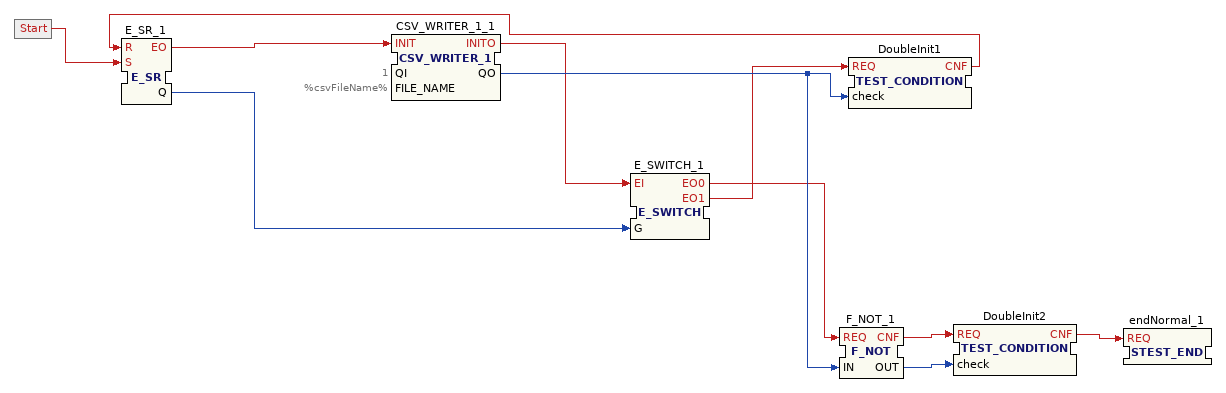
      FBS
        F_NOT_1 : F_NOT;
        E_SR_1 : E_SR;
        DoubleInit1 : TEST_CONDITION;
        CSV_WRITER_1_1 : CSV_WRITER_1(QI := 1, FILE_NAME := %csvFileName%);
        E_SWITCH_1 : E_SWITCH;
        endNormal_1 : STEST_END;
        DoubleInit2 : TEST_CONDITION;
      END_FBS
      EVENT_CONNECTIONS
        E_SWITCH_1.EO0 TO F_NOT_1.REQ;
        F_NOT_1.CNF TO DoubleInit2.REQ;
        DoubleInit1.CNF TO E_SR_1.R;
        E_SR_1.EO TO CSV_WRITER_1_1.INIT;
        E_SWITCH_1.EO1 TO DoubleInit1.REQ;
        CSV_WRITER_1_1.INITO TO E_SWITCH_1.EI;
        DoubleInit2.CNF TO endNormal_1.REQ;
        Start TO E_SR_1.S;
      END_CONNECTIONS
      DATA_CONNECTIONS
        CSV_WRITER_1_1.QO TO F_NOT_1.IN;
        F_NOT_1.OUT TO DoubleInit2.check;
        E_SR_1.Q TO E_SWITCH_1.G;
        CSV_WRITER_1_1.QO TO DoubleInit1.check;
      END_CONNECTIONS
    END_SUBAPPLICATION
    SUBAPPLICATION InitDeinitNoWrite
      EVENT_INPUT
        Start;
      END_EVENT
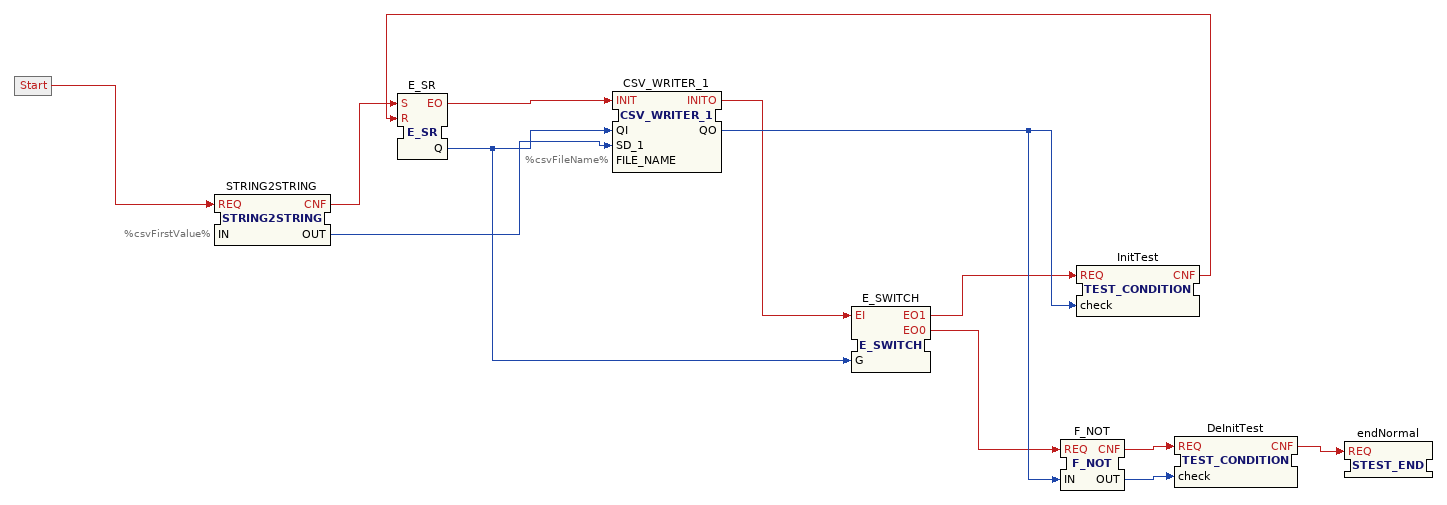
      FBS
        CSV_WRITER_1 : CSV_WRITER_1(FILE_NAME := %csvFileName%);
        InitTest : TEST_CONDITION;
        STRING2STRING : STRING2STRING(IN := %csvFirstValue%);
        DeInitTest : TEST_CONDITION;
        endNormal : STEST_END;
        F_NOT : F_NOT;
        E_SWITCH : E_SWITCH;
        E_SR : E_SR;
      END_FBS
      EVENT_CONNECTIONS
        E_SR.EO TO CSV_WRITER_1.INIT;
        CSV_WRITER_1.INITO TO E_SWITCH.EI;
        E_SWITCH.EO1 TO InitTest.REQ;
        STRING2STRING.CNF TO E_SR.S;
        F_NOT.CNF TO DeInitTest.REQ;
        DeInitTest.CNF TO endNormal.REQ;
        E_SWITCH.EO0 TO F_NOT.REQ;
        Start TO STRING2STRING.REQ;
        InitTest.CNF TO E_SR.R;
      END_CONNECTIONS
      DATA_CONNECTIONS
        E_SR.Q TO CSV_WRITER_1.QI;
        STRING2STRING.OUT TO CSV_WRITER_1.SD_1;
        CSV_WRITER_1.QO TO InitTest.check;
        CSV_WRITER_1.QO TO F_NOT.IN;
        F_NOT.OUT TO DeInitTest.check;
        E_SR.Q TO E_SWITCH.G;
      END_CONNECTIONS
    END_SUBAPPLICATION
    SUBAPPLICATION closeNotOpenedFile
      EVENT_INPUT
        Start;
      END_EVENT
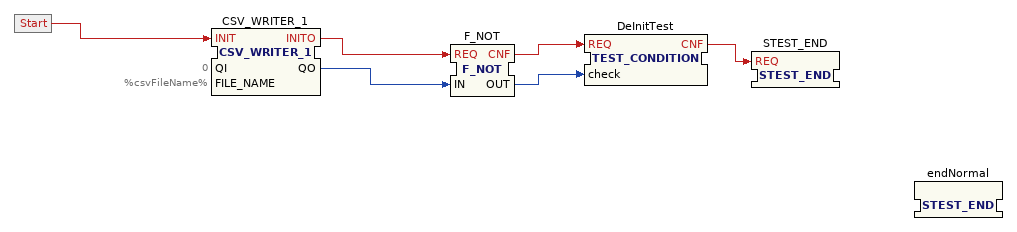
      FBS
        CSV_WRITER_1 : CSV_WRITER_1(QI := 0, FILE_NAME := %csvFileName%);
        DeInitTest : TEST_CONDITION;
        endNormal : STEST_END;
        F_NOT : F_NOT;
        STEST_END : STEST_END;
      END_FBS
      EVENT_CONNECTIONS
        F_NOT.CNF TO DeInitTest.REQ;
        CSV_WRITER_1.INITO TO F_NOT.REQ;
        Start TO CSV_WRITER_1.INIT;
        DeInitTest.CNF TO STEST_END.REQ;
      END_CONNECTIONS
      DATA_CONNECTIONS
        F_NOT.OUT TO DeInitTest.check;
        CSV_WRITER_1.QO TO F_NOT.IN;
      END_CONNECTIONS
    END_SUBAPPLICATION
    SUBAPPLICATION writeWithoutInit
      EVENT_INPUT
        Start;
      END_EVENT
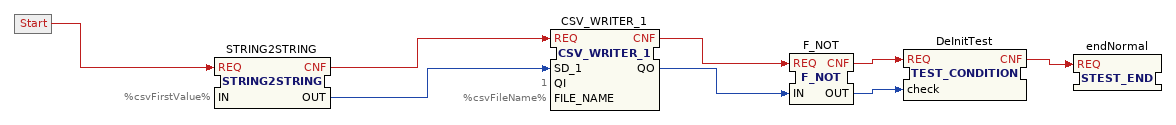
      FBS
        CSV_WRITER_1 : CSV_WRITER_1(QI := 1, FILE_NAME := %csvFileName%);
        STRING2STRING : STRING2STRING(IN := %csvFirstValue%);
        DeInitTest : TEST_CONDITION;
        endNormal : STEST_END;
        F_NOT : F_NOT;
      END_FBS
      EVENT_CONNECTIONS
        F_NOT.CNF TO DeInitTest.REQ;
        DeInitTest.CNF TO endNormal.REQ;
        Start TO STRING2STRING.REQ;
        STRING2STRING.CNF TO CSV_WRITER_1.REQ;
        CSV_WRITER_1.CNF TO F_NOT.REQ;
      END_CONNECTIONS
      DATA_CONNECTIONS
        STRING2STRING.OUT TO CSV_WRITER_1.SD_1;
        CSV_WRITER_1.QO TO F_NOT.IN;
        F_NOT.OUT TO DeInitTest.check;
      END_CONNECTIONS
    END_SUBAPPLICATION
    SUBAPPLICATION writeQIFalse
      EVENT_INPUT
        Start;
      END_EVENT
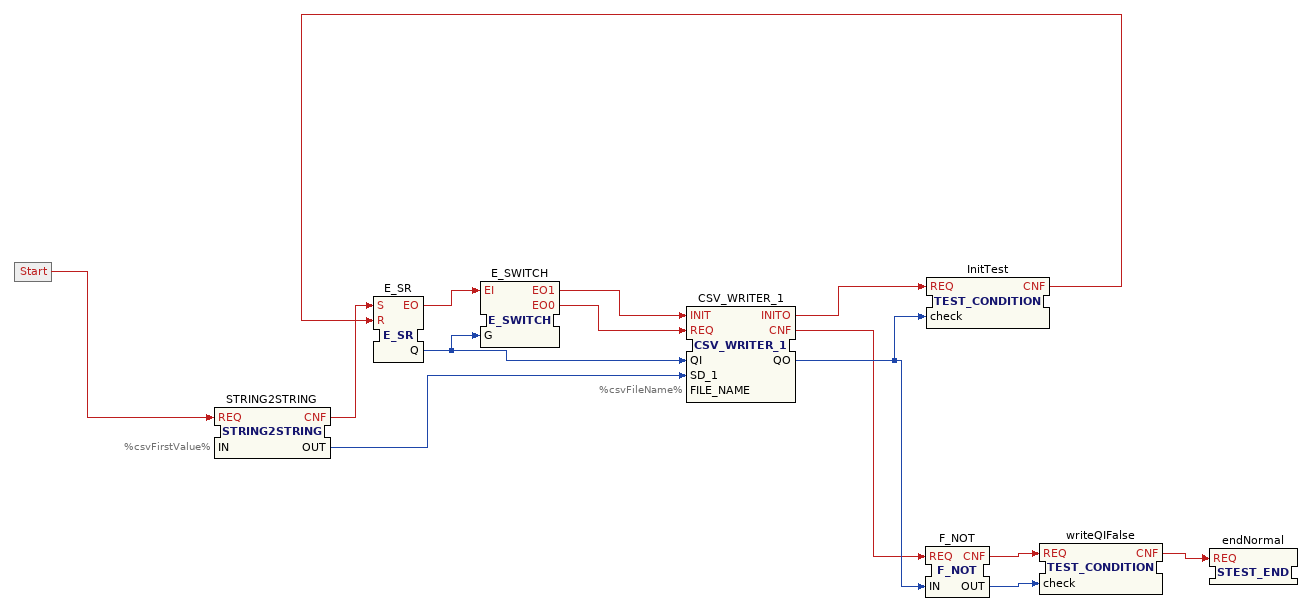
      FBS
        CSV_WRITER_1 : CSV_WRITER_1(FILE_NAME := %csvFileName%);
        InitTest : TEST_CONDITION;
        STRING2STRING : STRING2STRING(IN := %csvFirstValue%);
        writeQIFalse : TEST_CONDITION;
        endNormal : STEST_END;
        F_NOT : F_NOT;
        E_SR : E_SR;
        E_SWITCH : E_SWITCH;
      END_FBS
      EVENT_CONNECTIONS
        STRING2STRING.CNF TO E_SR.S;
        F_NOT.CNF TO writeQIFalse.REQ;
        writeQIFalse.CNF TO endNormal.REQ;
        Start TO STRING2STRING.REQ;
        CSV_WRITER_1.INITO TO InitTest.REQ;
        InitTest.CNF TO E_SR.R;
        E_SWITCH.EO1 TO CSV_WRITER_1.INIT;
        E_SWITCH.EO0 TO CSV_WRITER_1.REQ;
        E_SR.EO TO E_SWITCH.EI;
        CSV_WRITER_1.CNF TO F_NOT.REQ;
      END_CONNECTIONS
      DATA_CONNECTIONS
        E_SR.Q TO CSV_WRITER_1.QI;
        STRING2STRING.OUT TO CSV_WRITER_1.SD_1;
        CSV_WRITER_1.QO TO InitTest.check;
        CSV_WRITER_1.QO TO F_NOT.IN;
        F_NOT.OUT TO writeQIFalse.check;
        E_SR.Q TO E_SWITCH.G;
      END_CONNECTIONS
    END_SUBAPPLICATION
    SUBAPPLICATION NormalExecutionMultiple
      EVENT_INPUT
        Start;
      END_EVENT
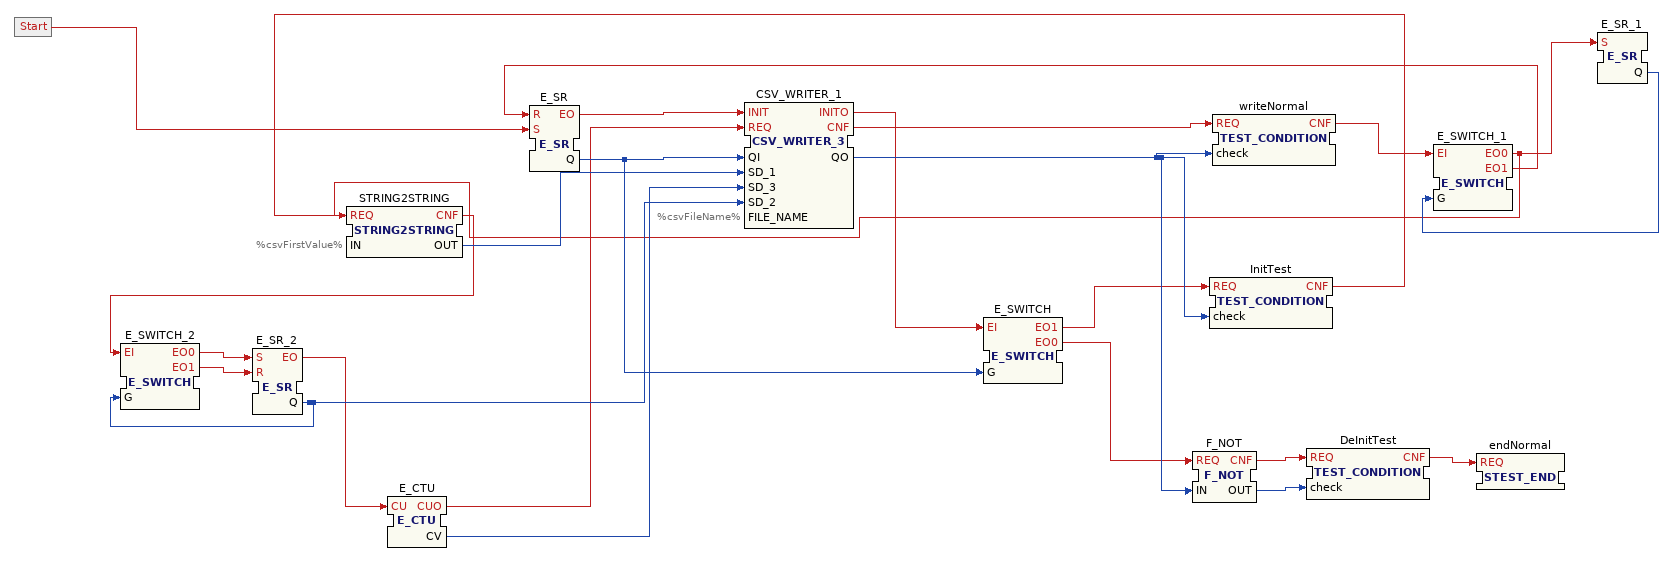
      FBS
        writeNormal : TEST_CONDITION;
        InitTest : TEST_CONDITION;
        STRING2STRING : STRING2STRING(IN := %csvFirstValue%);
        DeInitTest : TEST_CONDITION;
        endNormal : STEST_END;
        F_NOT : F_NOT;
        E_SWITCH : E_SWITCH;
        E_SR : E_SR;
        CSV_WRITER_1 : CSV_WRITER_3(FILE_NAME := %csvFileName%);
        E_SR_1 : E_SR;
        E_SWITCH_1 : E_SWITCH;
        E_SR_2 : E_SR;
        E_SWITCH_2 : E_SWITCH;
        E_CTU : E_CTU;
      END_FBS
      EVENT_CONNECTIONS
        E_SWITCH.EO1 TO InitTest.REQ;
        F_NOT.CNF TO DeInitTest.REQ;
        DeInitTest.CNF TO endNormal.REQ;
        E_SWITCH.EO0 TO F_NOT.REQ;
        E_SR.EO TO CSV_WRITER_1.INIT;
        CSV_WRITER_1.INITO TO E_SWITCH.EI;
        CSV_WRITER_1.CNF TO writeNormal.REQ;
        writeNormal.CNF TO E_SWITCH_1.EI;
        E_SWITCH_1.EO0 TO E_SR_1.S;
        E_SWITCH_1.EO1 TO E_SR.R;
        Start TO E_SR.S;
        InitTest.CNF TO STRING2STRING.REQ;
        E_SWITCH_1.EO0 TO STRING2STRING.REQ;
        STRING2STRING.CNF TO E_SWITCH_2.EI;
        E_SWITCH_2.EO0 TO E_SR_2.S;
        E_SWITCH_2.EO1 TO E_SR_2.R;
        E_CTU.CUO TO CSV_WRITER_1.REQ;
        E_SR_2.EO TO E_CTU.CU;
      END_CONNECTIONS
      DATA_CONNECTIONS
        F_NOT.OUT TO DeInitTest.check;
        E_SR.Q TO E_SWITCH.G;
        E_SR.Q TO CSV_WRITER_1.QI;
        STRING2STRING.OUT TO CSV_WRITER_1.SD_1;
        CSV_WRITER_1.QO TO InitTest.check;
        CSV_WRITER_1.QO TO F_NOT.IN;
        CSV_WRITER_1.QO TO writeNormal.check;
        E_SR_1.Q TO E_SWITCH_1.G;
        E_SR_2.Q TO E_SWITCH_2.G;
        E_CTU.CV TO CSV_WRITER_1.SD_3;
        E_SR_2.Q TO CSV_WRITER_1.SD_2;
      END_CONNECTIONS
    END_SUBAPPLICATION
    SUBAPPLICATION noNameFile
      EVENT_INPUT
        Start;
      END_EVENT
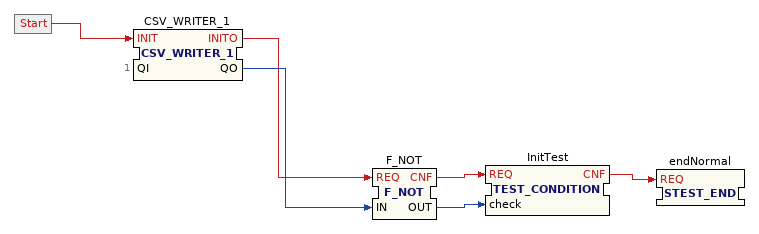
      FBS
        CSV_WRITER_1 : CSV_WRITER_1(QI := 1);
        InitTest : TEST_CONDITION;
        endNormal : STEST_END;
        F_NOT : F_NOT;
      END_FBS
      EVENT_CONNECTIONS
        F_NOT.CNF TO InitTest.REQ;
        InitTest.CNF TO endNormal.REQ;
        Start TO CSV_WRITER_1.INIT;
        CSV_WRITER_1.INITO TO F_NOT.REQ;
      END_CONNECTIONS
      DATA_CONNECTIONS
        CSV_WRITER_1.QO TO F_NOT.IN;
        F_NOT.OUT TO InitTest.check;
      END_CONNECTIONS
    END_SUBAPPLICATION
  END_APPLICATION
  APPLICATION MultiDevice
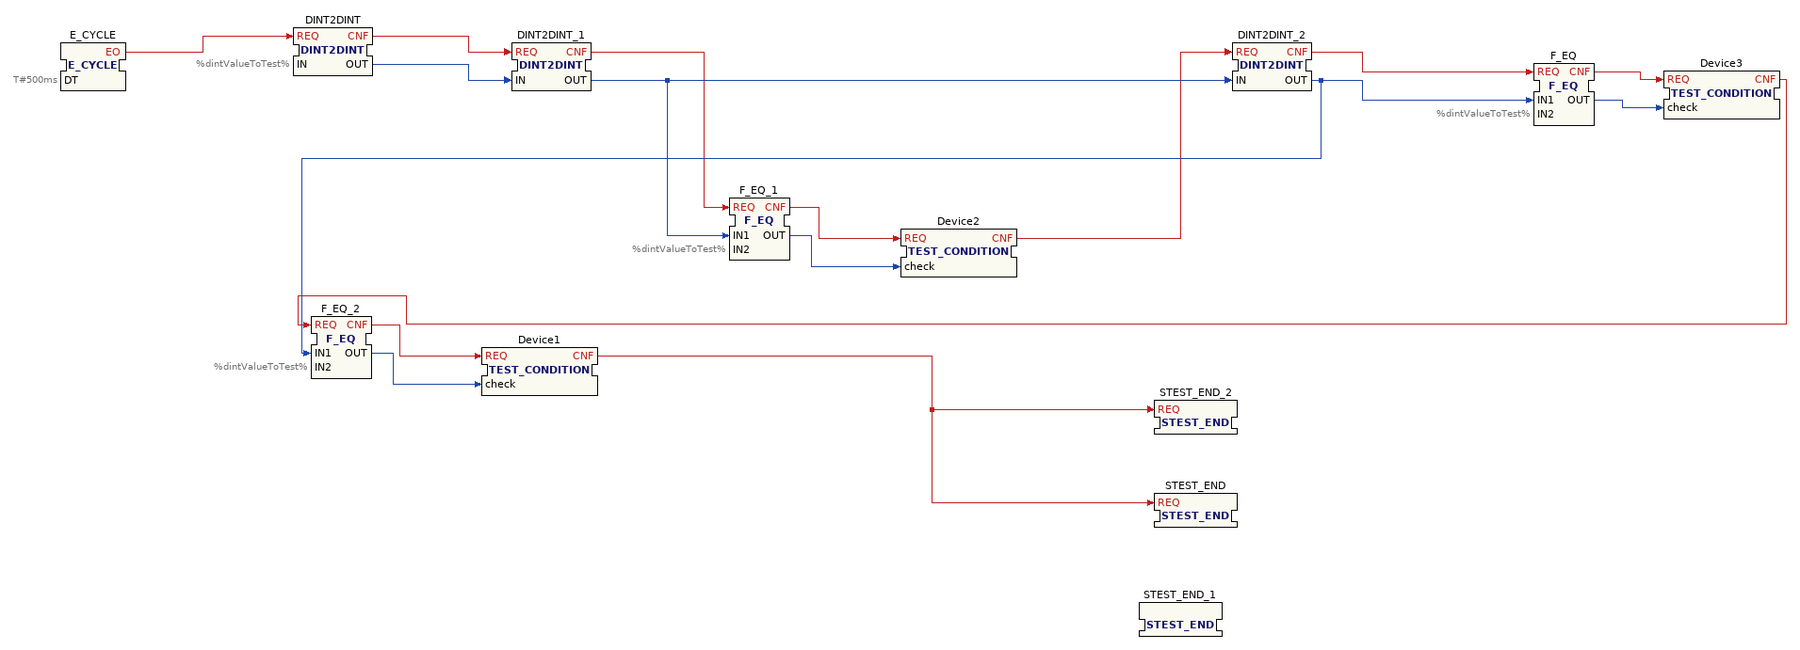
    FBS
      F_EQ_1 : F_EQ(IN2 := %dintValueToTest%);
      STEST_END : STEST_END;
      DINT2DINT_1 : DINT2DINT;
      DINT2DINT_2 : DINT2DINT;
      DINT2DINT : DINT2DINT(IN := %dintValueToTest%);
      Device3 : TEST_CONDITION;
      F_EQ : F_EQ(IN2 := %dintValueToTest%);
      Device2 : TEST_CONDITION;
      STEST_END_1 : STEST_END;
      E_CYCLE : E_CYCLE(DT := T#500ms);
      STEST_END_2 : STEST_END;
      F_EQ_2 : F_EQ(IN2 := %dintValueToTest%);
      Device1 : TEST_CONDITION;
    END_FBS
    EVENT_CONNECTIONS
      DINT2DINT.CNF TO DINT2DINT_1.REQ;
      F_EQ_1.CNF TO Device2.REQ;
      F_EQ.CNF TO Device3.REQ;
      DINT2DINT_2.CNF TO F_EQ.REQ;
      E_CYCLE.EO TO DINT2DINT.REQ;
      DINT2DINT_1.CNF TO F_EQ_1.REQ;
      Device2.CNF TO DINT2DINT_2.REQ;
      F_EQ_2.CNF TO Device1.REQ;
      Device3.CNF TO F_EQ_2.REQ;
      Device1.CNF TO STEST_END.REQ;
      Device1.CNF TO STEST_END_2.REQ;
    END_CONNECTIONS
    DATA_CONNECTIONS
      DINT2DINT_2.OUT TO F_EQ.IN1;
      DINT2DINT_1.OUT TO F_EQ_1.IN1;
      DINT2DINT_1.OUT TO DINT2DINT_2.IN;
      F_EQ_1.OUT TO Device2.check;
      F_EQ.OUT TO Device3.check;
      DINT2DINT.OUT TO DINT2DINT_1.IN;
      F_EQ_2.OUT TO Device1.check;
      DINT2DINT_2.OUT TO F_EQ_2.IN1;
    END_CONNECTIONS
  END_APPLICATION
  DEVICE DuT : FORTE_PC(MGR_ID := "localhost:61499" (* Device manager socket ID *))
    {SET_ATTRIBUTE(Profile, HOLOBLOC)}
    RESOURCE TimingTestRes : EMB_RES
      EVENT_CONNECTIONS
        START.COLD TO Timing.E_SR.S;
      END_CONNECTIONS
    END_RESOURCE
    RESOURCE Hard_Pass_Example : EMB_RES
      EVENT_CONNECTIONS
        START.COLD TO Hard_Pass_Example.BOOL2BOOL.REQ;
        START.WARM TO Hard_Pass_Example.BOOL2BOOL.REQ;
      END_CONNECTIONS
    END_RESOURCE
    RESOURCE Soft_Pass_Example : EMB_RES
      EVENT_CONNECTIONS
        START.COLD TO Soft_Pass_Example.F_MUX_2.REQ;
        START.WARM TO Soft_Pass_Example.F_MUX_2.REQ;
        START.COLD TO Soft_Pass_Example.BOOL2BOOL.REQ;
        START.WARM TO Soft_Pass_Example.BOOL2BOOL.REQ;
      END_CONNECTIONS
    END_RESOURCE
    RESOURCE Fail_Example : EMB_RES
      EVENT_CONNECTIONS
        START.COLD TO Fail_Example.BOOL2BOOL_1.REQ;
        START.WARM TO Fail_Example.BOOL2BOOL_1.REQ;
      END_CONNECTIONS
    END_RESOURCE
    RESOURCE DeInitCommFB : EMB_RES
      EVENT_CONNECTIONS
        START.COLD TO DeInitCommFB.E_SR_3.S;
        START.WARM TO DeInitCommFB.E_SR_3.S;
      END_CONNECTIONS
    END_RESOURCE
  END_DEVICE
  DEVICE Client : FORTE_PC(MGR_ID := "localhost:61499" (* Device manager socket ID *))
    {SET_ATTRIBUTE(Profile, HOLOBLOC)}
    RESOURCE simpleClientTest : EMB_RES
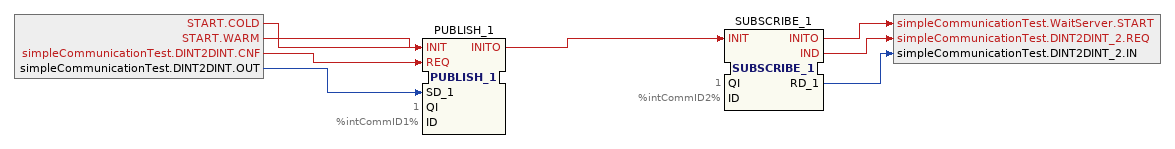
      FBS
        PUBLISH_1 : PUBLISH_1(QI := 1, ID := %intCommID1%);
        SUBSCRIBE_1 : SUBSCRIBE_1(QI := 1, ID := %intCommID2%);
      END_FBS
      EVENT_CONNECTIONS
        START.COLD TO PUBLISH_1.INIT;
        START.WARM TO PUBLISH_1.INIT;
        PUBLISH_1.INITO TO SUBSCRIBE_1.INIT;
        SUBSCRIBE_1.INITO TO simpleCommunicationTest.WaitServer.START;
        SUBSCRIBE_1.IND TO simpleCommunicationTest.DINT2DINT_2.REQ;
        simpleCommunicationTest.DINT2DINT.CNF TO PUBLISH_1.REQ;
      END_CONNECTIONS
      DATA_CONNECTIONS
        SUBSCRIBE_1.RD_1 TO simpleCommunicationTest.DINT2DINT_2.IN;
        simpleCommunicationTest.DINT2DINT.OUT TO PUBLISH_1.SD_1;
      END_CONNECTIONS
    END_RESOURCE
    RESOURCE multiDeviceStart : EMB_RES
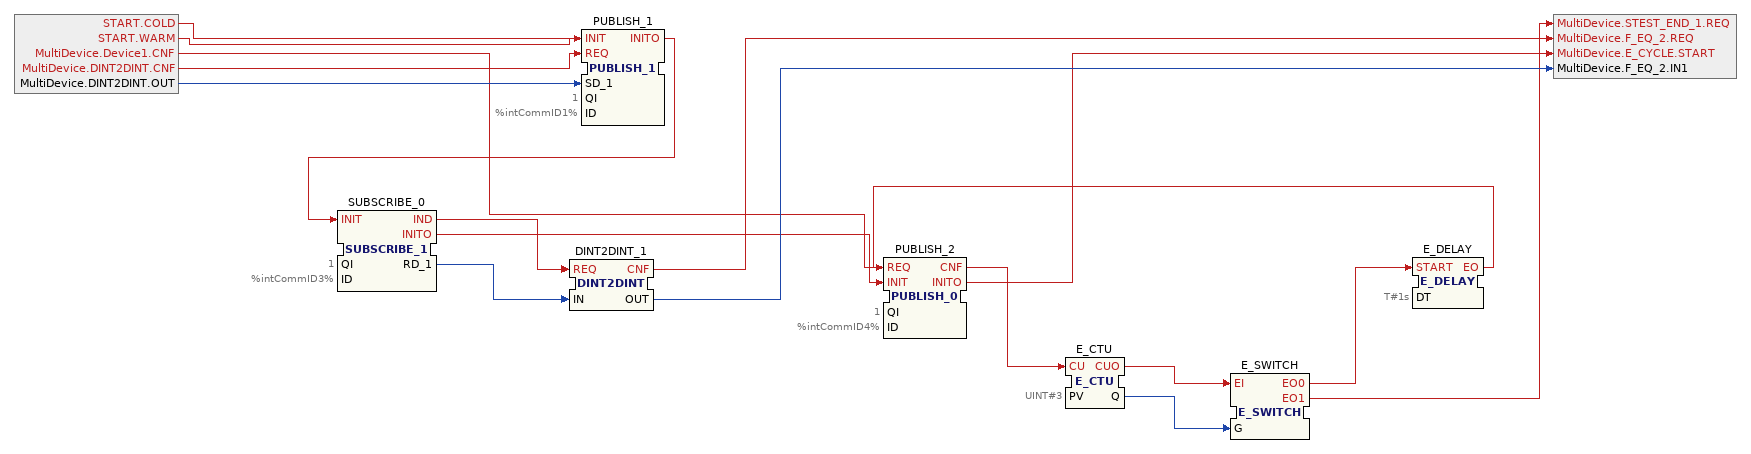
      FBS
        PUBLISH_1 : PUBLISH_1(QI := 1, ID := %intCommID1%);
        SUBSCRIBE_0 : SUBSCRIBE_1(QI := 1, ID := %intCommID3%);
        DINT2DINT_1 : DINT2DINT;
        E_DELAY : E_DELAY(DT := T#1s);
        PUBLISH_2 : PUBLISH_0(QI := 1, ID := %intCommID4%);
        E_CTU : E_CTU(PV := UINT#3);
        E_SWITCH : E_SWITCH;
      END_FBS
      EVENT_CONNECTIONS
        START.COLD TO PUBLISH_1.INIT;
        START.WARM TO PUBLISH_1.INIT;
        PUBLISH_1.INITO TO SUBSCRIBE_0.INIT;
        SUBSCRIBE_0.IND TO DINT2DINT_1.REQ;
        PUBLISH_2.CNF TO E_CTU.CU;
        E_CTU.CUO TO E_SWITCH.EI;
        E_SWITCH.EO0 TO E_DELAY.START;
        E_DELAY.EO TO PUBLISH_2.REQ;
        SUBSCRIBE_0.INITO TO PUBLISH_2.INIT;
        MultiDevice.Device1.CNF TO PUBLISH_2.REQ;
        E_SWITCH.EO1 TO MultiDevice.STEST_END_1.REQ;
        DINT2DINT_1.CNF TO MultiDevice.F_EQ_2.REQ;
        MultiDevice.DINT2DINT.CNF TO PUBLISH_1.REQ;
        PUBLISH_2.INITO TO MultiDevice.E_CYCLE.START;
      END_CONNECTIONS
      DATA_CONNECTIONS
        SUBSCRIBE_0.RD_1 TO DINT2DINT_1.IN;
        E_CTU.Q TO E_SWITCH.G;
        DINT2DINT_1.OUT TO MultiDevice.F_EQ_2.IN1;
        MultiDevice.DINT2DINT.OUT TO PUBLISH_1.SD_1;
      END_CONNECTIONS
    END_RESOURCE
  END_DEVICE
  DEVICE Server : FORTE_PC(MGR_ID := "localhost:61501" (* Device manager socket ID *))
    {SET_ATTRIBUTE(Profile, HOLOBLOC)}
    RESOURCE simpleServerTest : EMB_RES
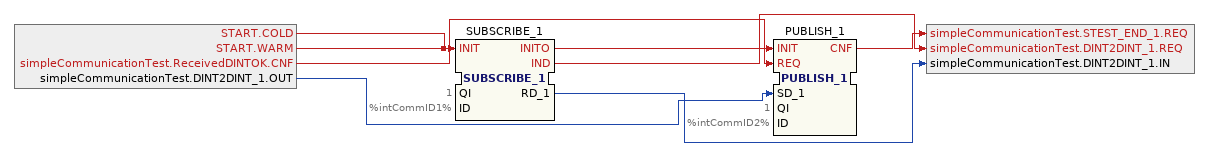
      FBS
        PUBLISH_1 : PUBLISH_1(QI := 1, ID := %intCommID2%);
        SUBSCRIBE_1 : SUBSCRIBE_1(QI := 1, ID := %intCommID1%);
      END_FBS
      EVENT_CONNECTIONS
        START.COLD TO SUBSCRIBE_1.INIT;
        START.WARM TO SUBSCRIBE_1.INIT;
        SUBSCRIBE_1.INITO TO PUBLISH_1.INIT;
        simpleCommunicationTest.ReceivedDINTOK.CNF TO PUBLISH_1.REQ;
        PUBLISH_1.CNF TO simpleCommunicationTest.STEST_END_1.REQ;
        SUBSCRIBE_1.IND TO simpleCommunicationTest.DINT2DINT_1.REQ;
      END_CONNECTIONS
      DATA_CONNECTIONS
        SUBSCRIBE_1.RD_1 TO simpleCommunicationTest.DINT2DINT_1.IN;
        simpleCommunicationTest.DINT2DINT_1.OUT TO PUBLISH_1.SD_1;
      END_CONNECTIONS
    END_RESOURCE
    RESOURCE multiDeviceEnd : EMB_RES
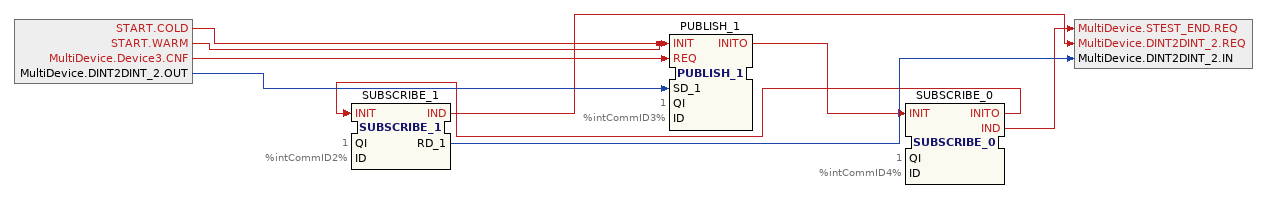
      FBS
        SUBSCRIBE_1 : SUBSCRIBE_1(QI := 1, ID := %intCommID2%);
        SUBSCRIBE_0 : SUBSCRIBE_0(QI := 1, ID := %intCommID4%);
        PUBLISH_1 : PUBLISH_1(QI := 1, ID := %intCommID3%);
      END_FBS
      EVENT_CONNECTIONS
        SUBSCRIBE_0.INITO TO SUBSCRIBE_1.INIT;
        START.COLD TO PUBLISH_1.INIT;
        START.WARM TO PUBLISH_1.INIT;
        PUBLISH_1.INITO TO SUBSCRIBE_0.INIT;
        MultiDevice.Device3.CNF TO PUBLISH_1.REQ;
        SUBSCRIBE_0.IND TO MultiDevice.STEST_END.REQ;
        SUBSCRIBE_1.IND TO MultiDevice.DINT2DINT_2.REQ;
      END_CONNECTIONS
      DATA_CONNECTIONS
        SUBSCRIBE_1.RD_1 TO MultiDevice.DINT2DINT_2.IN;
        MultiDevice.DINT2DINT_2.OUT TO PUBLISH_1.SD_1;
      END_CONNECTIONS
    END_RESOURCE
  END_DEVICE
  DEVICE CSVWriterTestDevice : FORTE_PC(MGR_ID := "localhost:61499" (* Device manager socket ID *))
    {SET_ATTRIBUTE(Profile, HOLOBLOC)}
    RESOURCE normalExecution : EMB_RES
      EVENT_CONNECTIONS
        START.COLD TO CSVWriterTests.NormalExecution.Start;
        START.WARM TO CSVWriterTests.NormalExecution.Start;
      END_CONNECTIONS
    END_RESOURCE
    RESOURCE openAndNoClose : EMB_RES
      EVENT_CONNECTIONS
        START.COLD TO CSVWriterTests.DontClose.Start;
        START.WARM TO CSVWriterTests.DontClose.Start;
      END_CONNECTIONS
    END_RESOURCE
    RESOURCE doubleInit : EMB_RES
      EVENT_CONNECTIONS
        START.COLD TO CSVWriterTests.DoubleInit.Start;
        START.WARM TO CSVWriterTests.DoubleInit.Start;
      END_CONNECTIONS
    END_RESOURCE
    RESOURCE initDeinitNoWrite : EMB_RES
      EVENT_CONNECTIONS
        START.COLD TO CSVWriterTests.InitDeinitNoWrite.Start;
        START.WARM TO CSVWriterTests.InitDeinitNoWrite.Start;
      END_CONNECTIONS
    END_RESOURCE
    RESOURCE closeNotOpened : EMB_RES
      EVENT_CONNECTIONS
        START.COLD TO CSVWriterTests.closeNotOpenedFile.Start;
        START.WARM TO CSVWriterTests.closeNotOpenedFile.Start;
      END_CONNECTIONS
    END_RESOURCE
    RESOURCE writeWithoutInit : EMB_RES
      EVENT_CONNECTIONS
        START.WARM TO CSVWriterTests.writeWithoutInit.Start;
        START.COLD TO CSVWriterTests.writeWithoutInit.Start;
      END_CONNECTIONS
    END_RESOURCE
    RESOURCE writeQIFalse : EMB_RES
      EVENT_CONNECTIONS
        START.COLD TO CSVWriterTests.writeQIFalse.Start;
        START.WARM TO CSVWriterTests.writeQIFalse.Start;
      END_CONNECTIONS
    END_RESOURCE
    RESOURCE normalExecutionMultiple : EMB_RES
      EVENT_CONNECTIONS
        START.COLD TO CSVWriterTests.NormalExecutionMultiple.Start;
        START.WARM TO CSVWriterTests.NormalExecutionMultiple.Start;
      END_CONNECTIONS
    END_RESOURCE
    RESOURCE noNameFile : EMB_RES
      EVENT_CONNECTIONS
        START.COLD TO CSVWriterTests.noNameFile.Start;
        START.WARM TO CSVWriterTests.noNameFile.Start;
      END_CONNECTIONS
    END_RESOURCE
  END_DEVICE
  DEVICE MiddleSystem : FORTE_PC(MGR_ID := "localhost:61500" (* Device manager socket ID *))
    {SET_ATTRIBUTE(Profile, HOLOBLOC)}
    RESOURCE multiDeviceMiddle : EMB_RES
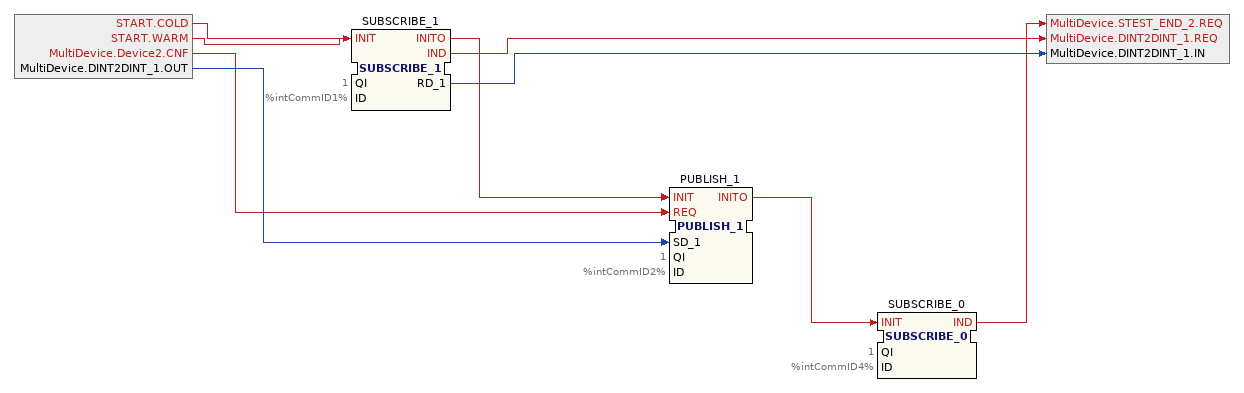
      FBS
        SUBSCRIBE_1 : SUBSCRIBE_1(QI := 1, ID := %intCommID1%);
        PUBLISH_1 : PUBLISH_1(QI := 1, ID := %intCommID2%);
        SUBSCRIBE_0 : SUBSCRIBE_0(QI := 1, ID := %intCommID4%);
      END_FBS
      EVENT_CONNECTIONS
        START.COLD TO SUBSCRIBE_1.INIT;
        START.WARM TO SUBSCRIBE_1.INIT;
        SUBSCRIBE_1.INITO TO PUBLISH_1.INIT;
        PUBLISH_1.INITO TO SUBSCRIBE_0.INIT;
        MultiDevice.Device2.CNF TO PUBLISH_1.REQ;
        SUBSCRIBE_0.IND TO MultiDevice.STEST_END_2.REQ;
        SUBSCRIBE_1.IND TO MultiDevice.DINT2DINT_1.REQ;
      END_CONNECTIONS
      DATA_CONNECTIONS
        SUBSCRIBE_1.RD_1 TO MultiDevice.DINT2DINT_1.IN;
        MultiDevice.DINT2DINT_1.OUT TO PUBLISH_1.SD_1;
      END_CONNECTIONS
    END_RESOURCE
  END_DEVICE
  MAPPINGS
    Timing.CSV_WRITER_1 ON DuT.TimingTestRes;
    Timing.E_SR ON DuT.TimingTestRes;
    Timing.E_SWITCH_2 ON DuT.TimingTestRes;
    Timing.Iterations ON DuT.TimingTestRes;
    Timing.FBNuTest ON DuT.TimingTestRes;
    Timing.STEST_END ON DuT.TimingTestRes;
    Timing.E_SWITCH ON DuT.TimingTestRes;
    Timing.E_StopWatch ON DuT.TimingTestRes;
    Soft_Pass_Example.NOT_ZERO ON DuT.Soft_Pass_Example;
    Soft_Pass_Example.F_NOT ON DuT.Soft_Pass_Example;
    Soft_Pass_Example.BOOL2BOOL ON DuT.Soft_Pass_Example;
    Soft_Pass_Example.STEST_END_0_1 ON DuT.Soft_Pass_Example;
    Soft_Pass_Example.F_MUX_2 ON DuT.Soft_Pass_Example;
    Fail_Example.BOOL2BOOL_1_1_1 ON DuT.Fail_Example;
    Fail_Example.BOOL2BOOL_1 ON DuT.Fail_Example;
    Fail_Example.BOOL2BOOL_1_1 ON DuT.Fail_Example;
    Fail_Example.STEST_END_0 ON DuT.Fail_Example;
    Fail_Example.SHOULD_FAIL_1 ON DuT.Fail_Example;
    Fail_Example.SHOULD_FAIL_2 ON DuT.Fail_Example;
    Fail_Example.SHOULD_NOT_FAIL ON DuT.Fail_Example;
    Hard_Pass_Example.STEST_END ON DuT.Hard_Pass_Example;
    Hard_Pass_Example.SHOULD_NOT_FAIL ON DuT.Hard_Pass_Example;
    Hard_Pass_Example.BOOL2BOOL ON DuT.Hard_Pass_Example;
    DeInitCommFB.E_SR ON DuT.DeInitCommFB;
    DeInitCommFB.E_SWITCH ON DuT.DeInitCommFB;
    DeInitCommFB.STEST_END ON DuT.DeInitCommFB;
    DeInitCommFB.PUBLISH_0 ON DuT.DeInitCommFB;
    DeInitCommFB.E_SWITCH_1 ON DuT.DeInitCommFB;
    DeInitCommFB.E_SR_1 ON DuT.DeInitCommFB;
    DeInitCommFB.E_SWITCH_2 ON DuT.DeInitCommFB;
    DeInitCommFB.E_SR_2 ON DuT.DeInitCommFB;
    DeInitCommFB.E_SR_3 ON DuT.DeInitCommFB;
    DeInitCommFB.E_SWITCH_3 ON DuT.DeInitCommFB;
    DeInitCommFB.PUBLISH_0_3 ON DuT.DeInitCommFB;
    DeInitCommFB.PUBLISH_0_2 ON DuT.DeInitCommFB;
    DeInitCommFB.PUBLISH_0_1 ON DuT.DeInitCommFB;
    simpleCommunicationTest.WaitServer ON Client.simpleClientTest;
    simpleCommunicationTest.ReturnetValueOK ON Client.simpleClientTest;
    simpleCommunicationTest.F_EQ_1 ON Server.simpleServerTest;
    simpleCommunicationTest.F_EQ ON Client.simpleClientTest;
    simpleCommunicationTest.STEST_END ON Client.simpleClientTest;
    simpleCommunicationTest.DINT2DINT ON Client.simpleClientTest;
    simpleCommunicationTest.ReceivedDINTOK ON Server.simpleServerTest;
    simpleCommunicationTest.DINT2DINT_1 ON Server.simpleServerTest;
    simpleCommunicationTest.DINT2DINT_2 ON Client.simpleClientTest;
    simpleCommunicationTest.STEST_END_1 ON Server.simpleServerTest;
    CSVWriterTests.NormalExecution ON CSVWriterTestDevice.normalExecution;
    CSVWriterTests.DontClose ON CSVWriterTestDevice.openAndNoClose;
    CSVWriterTests.DoubleInit ON CSVWriterTestDevice.doubleInit;
    CSVWriterTests.InitDeinitNoWrite ON CSVWriterTestDevice.initDeinitNoWrite;
    CSVWriterTests.closeNotOpenedFile ON CSVWriterTestDevice.closeNotOpened;
    CSVWriterTests.writeWithoutInit ON CSVWriterTestDevice.writeWithoutInit;
    CSVWriterTests.writeQIFalse ON CSVWriterTestDevice.writeQIFalse;
    CSVWriterTests.NormalExecutionMultiple ON CSVWriterTestDevice.normalExecutionMultiple;
    CSVWriterTests.noNameFile ON CSVWriterTestDevice.noNameFile;
    MultiDevice.DINT2DINT ON Client.multiDeviceStart;
    MultiDevice.DINT2DINT_1 ON MiddleSystem.multiDeviceMiddle;
    MultiDevice.F_EQ_1 ON MiddleSystem.multiDeviceMiddle;
    MultiDevice.Device2 ON MiddleSystem.multiDeviceMiddle;
    MultiDevice.STEST_END ON Server.multiDeviceEnd;
    MultiDevice.DINT2DINT_2 ON Server.multiDeviceEnd;
    MultiDevice.F_EQ ON Server.multiDeviceEnd;
    MultiDevice.Device3 ON Server.multiDeviceEnd;
    MultiDevice.E_CYCLE ON Client.multiDeviceStart;
    MultiDevice.STEST_END_2 ON MiddleSystem.multiDeviceMiddle;
    MultiDevice.STEST_END_1 ON Client.multiDeviceStart;
    MultiDevice.F_EQ_2 ON Client.multiDeviceStart;
    MultiDevice.Device1 ON Client.multiDeviceStart;
    Timing.Tracer1 ON DuT.TimingTestRes;
    Timing.Tracer2 ON DuT.TimingTestRes;
    Timing.E_SPLIT ON DuT.TimingTestRes;
    Timing.E_DELAY ON DuT.TimingTestRes;
  END_MAPPINGS
  SEGMENTS
    Ethernet : Ethernet;
  END_SEGMENTS
  LINKS
    Client => Ethernet;
    Server => Ethernet;
    MiddleSystem => Ethernet;
  END_LINKS
END_SYSTEM
